{attribute 'qualified_only'}
{attribute 'to_string'}
TYPE E_StepperHomingStates :
(
	Idle:=0,
	CheckIfEnabled,
	EnableAxis1,
	EnableAxis2,
	ResetAxis1,
	ResetAxis2,
	HomeSensorCheck,
	OutwardMotion,
	InwardMotion,
	OutwardCreep,
	WaitingForHalt,
	GettingCurrentPos,
	SettingHomePos,
	DisableAxis,
	WrapUp
)UINT := Idle
;
END_TYPE

(* stored: Version 1.1.0.1, ProductVersion 3.1.4024.12
   EnumerationTextList E_StepperHomingStates: Id {615bc563-79c1-4657-b4e2-ed52d9eb49c8} *)
